TYPE E_BPTMState :
(
	NewTarget := 1,
    WaitingForTransitionAssertion := 2,
    WaitingForFinalAssertion := 3,
    Transitioning := 4,
    CleaningUp := 5
);
END_TYPE

(* stored: Version 1.1.0.1, ProductVersion 3.1.4022.18
   DUT E_BPTMState: Id {768b40c8-623b-429d-9a70-34e6838c97c5} *)
